// TIA Portal V18 export
VAR_GLOBAL   // PLC tag table "Default tag table"
   FirstScan AT %M1.0 : Bool;
   DiagStatusUpdate AT %M1.1 : Bool;
   AlwaysTRUE AT %M1.2 : Bool;
   AlwaysFALSE AT %M1.3 : Bool;
END_VAR
